INTERFACE I_AsyncResponseManager

METHOD TryConvertResponseToAsyncResponseSessionData : BOOL
VAR_INPUT
	Response : I_ServerResponse;
	RetryDelayInMs : UDINT;
	Destination : REFERENCE TO I_AsyncResponseSessionData;
END_VAR
END_METHOD

METHOD PUBLIC TryHandleIncomingRequest : BOOL
VAR_INPUT
	Request : I_Request;
	Response : I_ServerResponse;
END_VAR
END_METHOD

END_INTERFACE

(* stored: Version 1.1.0.1, ProductVersion 3.1.4024.12
   Itf I_AsyncResponseManager: Id {abe05406-b7ab-4a25-a70f-e90409730aeb}
   Method TryConvertResponseToAsyncResponseSessionData: Id {32c68797-1e3f-4ba0-805b-b5c4e2259c26}
   Method TryHandleIncomingRequest: Id {dcc914a9-8a7f-4fe6-be9f-213c490e1a75} *)
